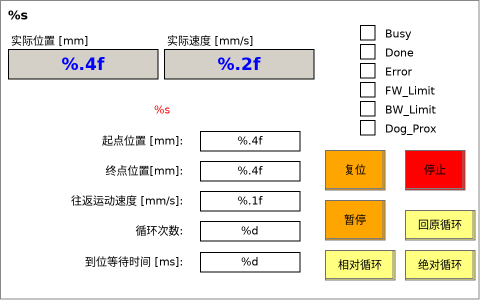
VISUALIZATION motionModuleP3  // 480x300
VAR_IN_OUT
	userData: motionModuleDataHMI;	
END_VAR
    Rectangle (36,126 150x30), "起点位置 [mm]:"
    Rectangle (36,156 150x30), "终点位置[mm]:"
    Rectangle (36,186 150x30), "往返运动速度 [mm/s]:"
    Rectangle (27,216 159x30), "循环次数:"
    Rectangle (8,49 150x30), "%.4f", text variable: userData.actualPos
    Rectangle (8,26 150x30), "实际位置 [mm]"
    Rectangle (164,49 150x30), "%.2f", text variable: userData.actualVel
    Rectangle (164,26 150x30), "实际速度 [mm/s]"
    Rectangle (12,100 300x20), "%s", text variable: userData.errTxt
    Rectangle (5,5 467x20), "%s", text variable: userData.nameTXT
    Rectangle (200,131 100x20), "%.4f", text variable: userData.loopFirstPoint
        OnMouseDown: write the text variable via Edit
    Rectangle (200,161 100x20), "%.4f", text variable: userData.loopSecondPoint
        OnMouseDown: write the text variable via Edit
    Rectangle (200,191 100x20), "%.1f", text variable: userData.loopGoVel
        OnMouseDown: write the text variable via Edit, min 0
    Rectangle (200,221 100x20), "%d", text variable: userData.loopCycle
        OnMouseDown: write the text variable via Edit, min 0
    Button (325,250 70x30), "相对循环", tooltip "Please keep pressing to trigger the relative motion loop", input disabled if: NOT userData.loopRelCondition OR NOT userData.ctrlModeCondition
        tap userData.loopRelGo
    Button (405,250 70x30), "绝对循环", tooltip "Please keep pressing to trigger the absolute motion loop", input disabled if: NOT userData.loopAbsCondition OR NOT userData.ctrlModeCondition
        tap userData.loopAbsGo
    Rectangle (27,247 159x30), "到位等待时间 [ms]:"
    Rectangle (200,252 100x20), "%d", text variable: userData.loopWatingTime
        OnMouseDown: write the text variable via Edit, min 0
    Button (405,150 60x40), "停止"
        tap userData.stop
    Button (325,150 60x40), "复位"
        tap userData.reset
    Rectangle (360,82 15x15), colour toggle: userData.forwardLimitSwitch
    Rectangle (360,101 15x15), colour toggle: userData.backwardsLimitSwitch
    Rectangle (360,120 15x15), colour toggle: userData.dogPointSwitch
    Rectangle (382,80 64x22), "FW_Limit"
    Rectangle (382,99 64x22), "BW_Limit"
    Rectangle (382,118 64x22), "Dog_Prox"
    Rectangle (360,25 15x15), colour toggle: userData.busy
    Rectangle (382,23 64x22), "Busy"
    Rectangle (382,42 64x22), "Done"
    Rectangle (382,61 64x22), "Error"
    Rectangle (360,44 15x15), colour toggle: userData.done
    Rectangle (360,63 15x15), colour toggle: userData.error
    Button (325,200 60x40), "暂停", colour toggle: userData.oPause, input disabled if: NOT userData.ctrlModeCondition
        tap userData.pauseB
    Button (405,210 70x30), "回原循环", tooltip "Please keep pressing to trigger the absolute motion loop", input disabled if: NOT userData.loopHomeToAbsCondition OR NOT userData.ctrlModeCondition
        tap userData.loopHomeToPosGo
END_VISUALIZATION

(* stored: Version 1.1.0.1, ProductVersion 3.1.4024.4
   Visu motionModuleP3: Id {7ceedbbc-a3e5-49c9-903a-96740654bffd} *)
